Fanuc KAREL source: kt00087.KL

-- PROVISIONAL review KL for V1013-1; original PC SHA256 bfb6bcb62e0d5f13424d49206e179ca2d37fa255b0b9815591682b497ad8c597
-- Incomplete behavior may be omitted. Consult companion uncertainty JSON. Do not deploy.
PROGRAM KT00087
%NOLOCKGROUP
VAR
  OUT : INTEGER
-- UNRESOLVED_DECL Y1 type=002018
-- UNRESOLVED_DECL H2 type=002017
BEGIN
  -- UNRESOLVED_PC offsets 5-19; opcodes 2E,22,9D,33,B2
  -- UNRESOLVED_PC offsets 24-38; opcodes 2E,22,9D,33,B4
  -- UNRESOLVED_PC offsets 43-68; opcodes 22,9D,33,B1,22,9D,33,B3,54,23
  -- UNRESOLVED_PC offsets 73-77; opcodes 7F
END KT00087
